FUNCTION_BLOCK FB_BottleFiller_Test EXTENDS FB_TestSuite

VAR	
END_VAR

TurningOnTheValveIfValveIsEmpty();

METHOD SettingThePressure
VAR_INPUT
END_VAR
END_METHOD

METHOD TurningOnTheValveIfValveIsEmpty
VAR_INPUT
END_VAR
VAR
	fbBottleFiller : FB_BottleFiller;
	fbBottle : FB_BottleFiller;
END_VAR
TEST('TurningOnTheValveIfValveIsEmpty');

fbBottleFiller.bisTankEmpty := TRUE;
fbBottleFiller.StartFilling();
AssertTrue(Condition := fbBottleFiller.bFilling,
		   Message := 'Tank is not Empty');

fbBottleFiller.bLevelSensor := TRUE;
fbBottleFiller.StopFilling();

AssertFalse(Condition := fbBottleFiller.bFilling, 
			 Message := 'Tank is filling');
TEST_FINISHED();
END_METHOD

END_FUNCTION_BLOCK

(* stored: Version 1.1.0.1, ProductVersion 3.1.4024.16
   POU FB_BottleFiller_Test: Id {ee18a254-76ee-4cdc-a982-a7ec347d4bf4}, SpecialFunc None
   Method SettingThePressure: Id {c9e7dafd-786c-4278-98e3-3c594573f1e3}
   Method TurningOnTheValveIfValveIsEmpty: Id {4769dfd1-bd24-40b1-a8cd-ee27c407d8a7} *)
